INTERFACE I_Handler

METHOD handle : BOOL
VAR_INPUT
	request	:	STRING;
END_VAR
END_METHOD

METHOD setNext : BOOL
VAR_INPUT
	h	: I_Handler;
END_VAR
END_METHOD

END_INTERFACE

(* stored: Version 1.1.0.1, ProductVersion 3.1.4024.12
   Itf I_Handler: Id {5ca18d04-dcd9-04d4-04ce-4393759814d6}
   Method handle: Id {cf4379a9-e6b4-0a0e-0fa6-a0d0afe5ba8e}
   Method setNext: Id {bf74a296-1b70-0576-1d79-66e046376d94} *)
